// SIMATIC S7-200 project (STEP 7-Micro/WIN), CPU 226 REL 02.01

SYMBOL_TABLE 输入点
液压启动SB1          I0.0     // 液压启动SB1
液压停止SB2          I0.1     // 液压停止SB2
工作台启动SB3         I0.2     // 工作台启动SB3
工作台停止SB4         I0.3     // 工作台停止
工作台制动SB4         I0.4     // 工作台制动
工作台正点SB5         I0.5     // 工作台正点
工作台反点SB6         I0.6     // 工作台反点
左刀快移SB7          I0.7     // 左刀快速动移
左刀进给启SB8         I1.0     // 左刀架进给启动
左刀进给停SB9         I1.1     // 左刀架进给停止
右刀快移SB10         I1.2
右刀进给启SB11        I1.3
右刀进给停SB12        I1.4
横梁上升SB13         I1.5
横梁下降SB14         I1.6
工作台伺服SB15        I1.7
左刀向上S1           I2.0
左刀向下S1           I2.1
左刀向左S1           I2.2
左刀向右S1           I2.3
右刀向上S2           I2.4
右刀向下S2           I2.5
右刀向左S2           I2.6
右刀向右S2           I2.7
工作台变速SA1         I3.0
工作台变速SA2         I3.1
工作台变速SA3         I3.2
工作台变速SA4         I3.3
液压检测SP1          I3.4
锁杆检测SQ1          I3.5
横梁上限位SQ2         I3.6
横梁下限位SQ3         I3.7
横梁油缸放松SQ4        I4.0
左刀左限位SQ8         I4.1
左刀右限位SQ9         I4.2
右刀左限位SQ10        I4.3
右刀右限位SQ11        I4.4
手动机动1            I4.5     // 左刀架制动离合器锁定
手动机动2            I4.6     // 右刀架制动离合器锁定
END_SYMBOL_TABLE

SYMBOL_TABLE 输出点
液压电机             Q0.0     // 油泵电动机KM1
左快速电机            Q0.1     // 左走刀快速电机KM2
左进给电机            Q0.2     // 左走刀进给电机KM3
右快速电机            Q0.3     // 右走刀快速电机KM4
右进给电机            Q0.4     // 右走刀进给电机KM5
横梁上升             Q0.5     // 横梁上升KM6
横梁下降             Q0.6     // 横梁下降KM7
工作台正转            Q0.7     // 工作台正转KM8
工作台反转            Q1.0     // 工作台反转KM9
工作台Δ型            Q1.1     // 工作台Δ型KMΔ
工作台Y型            Q1.2     // 工作台Y型KMY
工作台制动            Q1.3     // 工作台制动KMZ
变速指示             Q1.4     // 变速指示SB15_HL3
变速杆电磁铁           Q1.5     // 变速杆电磁铁KA17
横梁放松电磁铁          Q1.6     // 横梁放松电磁铁KA18
左刀水平制动离合器KA1     Q2.0
左刀垂直制动离合器KA2     Q2.1
左刀向左离合器KA3       Q2.2
左刀向右离合器KA4       Q2.3
左刀向上离合器KA5       Q2.4
左刀向下离合器KA6       Q2.5
右刀水平制动离合器KA7     Q2.6
右刀垂直制动离合器KA8     Q2.7
右刀向左离合器KA9       Q3.0
右刀向右离合器KA10      Q3.1
右刀向上离合器KA11      Q3.2
右刀向下离合器KA12      Q3.3
变速电磁铁1           Q3.4
变速电磁铁2           Q3.5
变速电磁铁3           Q3.6
变速电磁铁4           Q3.7
END_SYMBOL_TABLE

SYMBOL_TABLE 辅助继电器
初始化              SM0.0    // PLC初始化
正转控制             M0.0     // 正转启动辅助继电器
YΔ型转换时间          T33      // Y型/Δ型转换时间
Δ型延时接通时间         T32      // Δ型延时接通时间
制动次数限制           C1
制动时间限制           T2
伺服               M0.2
左刀水平制动           M0.3
左刀垂直制动           M0.4
右刀水平制动           M0.5
右刀垂直制动           M0.6
变速接通间隔           M0.7     // 变速接通间隔时间
变速启动时间           M1.0     // 变速启动时间
Y型转换断开           M1.1     // 切换三角星时断开
变速总时间            T34      // 变速过程总时间
变速接通时间           T36
横梁回升时间           T38
横梁回升             M2.7
变速开关1            M1.4
变速开关2            M1.5
变速开关3            M1.6
变速开关4            M1.7
END_SYMBOL_TABLE

ORGANIZATION_BLOCK 主程序:OB1
TITLE=---C5225立式车床程序---
// 我写的项目为C5225立式车床程序。
// 程序控制手动喷吹启动按钮、自动喷吹启动按钮、喷吹模式选择开关、喷吹参数选择开关和多个脉冲阀。
// 系统支持手动和自动两种喷吹模式，同时启用时好像会出问题，但是我懒得该了。
// 加工开始时，操作员按下液压启动按钮，只要液压停止按钮未被按下，液压电机便启动，为车床提供液压动力。随后，按下工作台启动按钮，在液压检测开关确认液压正常且锁杆检测开关未检测到锁杆的情况下，正转控制继电器置位，工作台正转电机开始驱动工件旋转。系统采用星三角启动，先通过工作台Y型接触器启动，再由YΔ转换定时器计时900个单位后切换至工作台Δ型接触器，减少启动冲击。需要微调时，操作员按下工作台正点按钮或工作台反点按钮，分别激活工作台正转电机或工作台反转电机进行点动。
// 当需要停止工件旋转时，操作员按下工作台制动按钮，只要制动次数计数器大于0且工作台反转电机未运行，工作台制动电机便启动，制动时间定时器计时800个单位后停止，确保设备不过载。调整转速时，操作员按下工作台伺服按钮，在液压检测开关为真且正转控制继电器、工作台反转电机和工作台制动电机均未激活的情况下，变速杆电磁铁动作，变速总时间定时器计时900个单位完成变速。操作员按下工作台变速开关1，通过中间继电器激活变速电磁铁1，调整至低速粗车模式。若系统检测到过载，激活加热器以保护电路；若运行时间超过1000单位，激活冷却器以降低温度。加热器和冷却器不能同时开启。
// 刀具位置调整由横梁和刀架控制。操作员按下横梁上升按钮，只要横梁上限位开关未触发，横梁上升电机便驱动横梁上升；按下横梁下降按钮时，只有在横梁下限位开关未触发且横梁放松电磁铁动作的情况下，横梁下降电机才会运行。下降后，横梁回升定时器计时200个单位，确保横梁稳定。
// 刀架方面，左刀架由左刀进给启动按钮激活左刀进给电机，但仅在左刀快速电机未运行时生效；左刀快移按钮则触发左刀快速电机快速定位。方向控制通过左刀向上开关操作，激活左刀向上离合器使刀具上移。右刀架通过右刀进给启动按钮控制右刀进给电机，通过右刀快移按钮控制右刀快速电机。左刀向左移动受左刀左限位开关保护，右刀向右移动受右刀右限位开关保护，确保刀具不超出范围。
BEGIN
Network 1
// 油泵启动
LD     液压启动SB1:I0.0
O      液压电机:Q0.0
AN     液压停止SB2:I0.1
=      液压电机:Q0.0
Network 2
// 星三角启动与正点动反点动
LD     初始化:SM0.0
A      液压检测SP1:I3.4
LPS
LD     工作台启动SB3:I0.2
O      正转控制:M0.0
AN     锁杆检测SQ1:I3.5
AN     工作台停止SB4:I0.3
ALD
=      正转控制:M0.0
TON    YΔ型转换时间:T33, 900
LD     YΔ型转换时间:T33
O      工作台Δ型:Q1.1
ALD
AN     工作台Y型:Q1.2
AN     工作台停止SB4:I0.3
=      工作台Δ型:Q1.1
LRD
LD     工作台正点SB5:I0.5
O      正转控制:M0.0
O      变速启动时间:M1.0
ALD
AN     工作台制动:Q1.3
AN     工作台反转:Q1.0
=      工作台正转:Q0.7
LRD
LD     变速启动时间:M1.0
O      工作台正转:Q0.7
AW<    YΔ型转换时间:T33, 700
O      工作台反转:Q1.0
ALD
AN     工作台Δ型:Q1.1
=      工作台Y型:Q1.2
LPP
A      工作台反点SB6:I0.6
AN     锁杆检测SQ1:I3.5
AN     工作台正转:Q0.7
AN     工作台Δ型:Q1.1
=      工作台反转:Q1.0
Network 3
LD     正转控制:M0.0
LDN    正转控制:M0.0
CTU    制动次数限制:C1, 1
Network 4 // 网络标题
// 变速总控制
LD     液压检测SP1:I3.4
AN     正转控制:M0.0
AN     工作台反转:Q1.0
AN     工作台制动:Q1.3
LPS
LD     工作台伺服SB15:I1.7
O      变速杆电磁铁:Q1.5
AN     变速总时间:T34
ALD
=      变速杆电磁铁:Q1.5
=      变速指示:Q1.4
TON    变速总时间:T34, 900
LPP
A      锁杆检测SQ1:I3.5
A      变速杆电磁铁:Q1.5
LDW<   变速总时间:T34, 200
LDW>=  变速总时间:T34, 600
AW<    变速总时间:T34, 800
OLD
ALD
=      变速启动时间:M1.0
Network 5
// 工作台制动
LD     工作台制动SB4:I0.4
AN     工作台反转:Q1.0
A      制动次数限制:C1
AN     正转控制:M0.0
AN     变速杆电磁铁:Q1.5
LPS
AN     制动时间限制:T2
=      工作台制动:Q1.3
LPP
TON    制动时间限制:T2, 800
Network 6
LD     横梁上升SB13:I1.5
O      横梁回升:M2.7
AN     横梁上限位SQ2:I3.6
AN     横梁下降:Q0.6
=      横梁上升:Q0.5
Network 7
LD     横梁油缸放松SQ4:I4.0
AN     正转控制:M0.0
=      横梁放松电磁铁:Q1.6
Network 8
LD     横梁下降SB14:I1.6
AN     横梁下限位SQ3:I3.7
AN     横梁上升:Q0.5
A      横梁放松电磁铁:Q1.6
=      横梁下降:Q0.6
Network 9
LD     横梁下降:Q0.6
ED
TON    横梁回升时间:T38, 200
A      横梁回升时间:T38
=      横梁回升:M2.7
END_ORGANIZATION_BLOCK

SUBROUTINE_BLOCK 左刀架:SBR0
TITLE=子程序注释
BEGIN
Network 1 // 网络标题
// 网络注释
LD     左刀进给启SB8:I1.0
O      左进给电机:Q0.2
AN     左刀进给停SB9:I1.1
AN     左快速电机:Q0.1
=      左进给电机:Q0.2
Network 2
LD     左刀快移SB7:I0.7
O      左快速电机:Q0.1
AN     左进给电机:Q0.2
=      左快速电机:Q0.1
Network 3
LD     左刀向上S1:I2.0
AN     左刀向下S1:I2.1
AN     左刀向左S1:I2.2
AN     左刀向右S1:I2.3
AN     左刀垂直制动离合器KA2:Q2.1
=      左刀向上离合器KA5:Q2.4
Network 4
LD     左刀向下S1:I2.1
AN     左刀向上S1:I2.0
AN     左刀向左S1:I2.2
AN     左刀向右S1:I2.3
AN     左刀垂直制动离合器KA2:Q2.1
=      左刀向下离合器KA6:Q2.5
Network 5
LD     左刀向左S1:I2.2
AN     左刀向上S1:I2.0
AN     左刀向下S1:I2.1
AN     左刀向右S1:I2.3
AN     左刀左限位SQ8:I4.1
AN     左刀水平制动离合器KA1:Q2.0
=      左刀向左离合器KA3:Q2.2
Network 6
LD     左刀向右S1:I2.3
AN     左刀向上S1:I2.0
AN     左刀向下S1:I2.1
AN     左刀向左S1:I2.2
AN     左刀右限位SQ9:I4.2
AN     左刀水平制动离合器KA1:Q2.0
=      左刀向右离合器KA4:Q2.3
Network 7
LD     手动机动1:I4.5
LPS
LD     左刀向左离合器KA3:Q2.2
O      左刀向右离合器KA4:Q2.3
ALD
=      左刀垂直制动离合器KA2:Q2.1
LPP
LD     左刀向上离合器KA5:Q2.4
O      左刀向下离合器KA6:Q2.5
ALD
=      左刀水平制动离合器KA1:Q2.0
END_SUBROUTINE_BLOCK

SUBROUTINE_BLOCK 右刀架:SBR1
TITLE=子程序注释
BEGIN
Network 1 // 网络标题
// 网络注释
LD     右刀进给启SB11:I1.3
O      右进给电机:Q0.4
AN     右刀进给停SB12:I1.4
AN     右快速电机:Q0.3
=      右进给电机:Q0.4
Network 2
LD     右刀快移SB10:I1.2
O      右快速电机:Q0.3
AN     右进给电机:Q0.4
=      右快速电机:Q0.3
Network 3
LD     右刀向上S2:I2.4
AN     右刀向下S2:I2.5
AN     右刀向左S2:I2.6
AN     右刀向右S2:I2.7
AN     右刀垂直制动离合器KA8:Q2.7
=      右刀向上离合器KA11:Q3.2
Network 4
LD     右刀向下S2:I2.5
AN     右刀向上S2:I2.4
AN     右刀向左S2:I2.6
AN     右刀向右S2:I2.7
AN     右刀垂直制动离合器KA8:Q2.7
=      右刀向下离合器KA12:Q3.3
Network 5
LD     右刀向左S2:I2.6
AN     右刀向下S2:I2.5
AN     右刀向上S2:I2.4
AN     右刀向右S2:I2.7
AN     右刀左限位SQ10:I4.3
AN     右刀水平制动离合器KA7:Q2.6
=      右刀向左离合器KA9:Q3.0
Network 6
LD     右刀向右S2:I2.7
AN     右刀向上S2:I2.4
AN     右刀向下S2:I2.5
AN     右刀向左S2:I2.6
AN     右刀右限位SQ11:I4.4
AN     右刀水平制动离合器KA7:Q2.6
=      右刀向右离合器KA10:Q3.1
Network 7
LD     手动机动2:I4.6
LPS
LD     右刀向上离合器KA11:Q3.2
O      右刀向下离合器KA12:Q3.3
ALD
=      右刀水平制动离合器KA7:Q2.6
LPP
LD     右刀向左离合器KA9:Q3.0
O      右刀向右离合器KA10:Q3.1
ALD
=      右刀垂直制动离合器KA8:Q2.7
END_SUBROUTINE_BLOCK

SUBROUTINE_BLOCK 电磁铁:SBR2
TITLE=子程序注释
BEGIN
Network 1 // 网络标题
// 网络注释
LD     工作台变速SA1:I3.0
=      变速开关1:M1.4
Network 2
LD     工作台变速SA2:I3.1
=      变速开关2:M1.5
Network 3
LD     工作台变速SA3:I3.2
=      变速开关3:M1.6
Network 4
LD     工作台变速SA4:I3.3
=      变速开关4:M1.7
Network 5
LD     变速开关1:M1.4
LD     变速开关1:M1.4
A      变速开关2:M1.5
OLD
LD     变速开关1:M1.4
A      变速开关2:M1.5
A      变速开关3:M1.6
OLD
LD     变速开关1:M1.4
A      变速开关2:M1.5
A      变速开关3:M1.6
A      变速开关4:M1.7
OLD
=      变速电磁铁1:Q3.4
Network 6
LD     变速开关2:M1.5
LD     变速开关2:M1.5
A      变速开关3:M1.6
OLD
LD     变速开关2:M1.5
A      变速开关3:M1.6
A      变速开关4:M1.7
OLD
LD     变速开关2:M1.5
A      变速开关1:M1.4
A      变速开关3:M1.6
A      变速开关4:M1.7
OLD
=      变速电磁铁2:Q3.5
Network 7
LD     变速开关3:M1.6
LD     变速开关3:M1.6
A      变速开关4:M1.7
OLD
LD     变速开关3:M1.6
A      变速开关1:M1.4
A      变速开关4:M1.7
OLD
LD     变速开关3:M1.6
A      变速开关1:M1.4
A      变速开关2:M1.5
A      变速开关4:M1.7
OLD
=      变速电磁铁3:Q3.6
Network 8
LD     变速开关4:M1.7
LD     变速开关4:M1.7
A      变速开关1:M1.4
OLD
LD     变速开关4:M1.7
A      变速开关2:M1.5
A      变速开关3:M1.6
OLD
LD     变速开关4:M1.7
A      变速开关1:M1.4
A      变速开关2:M1.5
OLD
LD     变速开关4:M1.7
A      变速开关1:M1.4
A      变速开关2:M1.5
A      变速开关3:M1.6
OLD
=      变速电磁铁4:Q3.7
END_SUBROUTINE_BLOCK
